(* IEC 61131-3 sources: sphere-usecases/power-hydro/implementations/openplc/st, 2 files *)

(* ---- ps_hydro_controller.st ---- *)
(*
 * SPHERE Power Systems - Generic Hydro Station Controller
 * IEC 61131-3 Structured Text for OpenPLC (matiec compatible)
 *
 * Control state machine for hydro power generation:
 *   IDLE -> STARTUP -> RUNNING -> SHUTDOWN -> IDLE
 *                  \-> TRIPPED (on any trip) -> IDLE (after reset)
 *
 * I/O Mapping (configured in OpenPLC web interface):
 *   HMI Inputs:
 *     in_Start_Cmd -> %IX0.0
 *     in_Stop_Cmd -> %IX0.1
 *     in_Reset_Cmd -> %IX0.2
 *     in_Mode_Auto -> %IX0.3
 *     in_Run_Enable -> %IX0.4
 *     in_Power_Setpoint -> %IW60
 *
 *   Process Inputs from Simulator (via bridge):
 *     in_Gate_Pos -> %IW70
 *     in_Res_Level -> %IW71
 *     in_Head -> %IW72
 *     in_Flow -> %IW73
 *     in_Pressure -> %IW74
 *     in_Speed_Pct -> %IW75
 *     in_Freq_Hz -> %IW76
 *     in_Power_MW -> %IW77
 *     in_Breaker_Sts -> %IX2.0
 *     in_Spill_Sts -> %IX2.1
 *
 *   Actuator Outputs to Simulator (via bridge):
 *     out_Gate_Cmd -> %QW100
 *     out_Power_Setpoint -> %QW101
 *     out_Breaker_Cmd -> %QX5.0
 *     out_Spill_Cmd -> %QX5.1
 *
 *   State Outputs to HMI:
 *     out_State_Idle -> %QX7.0
 *     out_State_Startup -> %QX7.1
 *     out_State_Running -> %QX7.2
 *     out_State_Shutdown -> %QX7.3
 *     out_State_Tripped -> %QX7.4
 *     out_Permissives_Ready -> %QX7.5
 *
 *   Trip Outputs:
 *     out_Trip_Overspeed -> %QX8.0
 *     out_Trip_Overpressure -> %QX8.1
 *     out_Trip_LowHead -> %QX8.2
 *     out_Trip_Manual -> %QX8.3
 *
 *   Alarm Outputs:
 *     out_Alarm_GateMismatch -> %QX9.0
 *     out_Alarm_BreakerMismatch -> %QX9.1
 *     out_Alarm_LowLevel -> %QX9.2
 *)

PROGRAM HydroController
  VAR_INPUT
    (* HMI Inputs *)
    in_Start_Cmd : BOOL;              (* Start pushbutton *)
    in_Stop_Cmd : BOOL;               (* Stop pushbutton *)
    in_Reset_Cmd : BOOL;              (* Trip reset pushbutton *)
    in_Mode_Auto : BOOL;              (* Auto mode enable *)
    in_Run_Enable : BOOL;             (* Run permissive *)
    in_Power_Setpoint : INT;          (* 0-1000 = 0-100 MW *)

    (* Process Inputs from Simulator *)
    in_Gate_Pos : INT;                (* Gate position 0-1000 = 0-100% *)
    in_Res_Level : INT;               (* Reservoir level 0-3000 = 0-30.00 m *)
    in_Head : INT;                    (* Head 0-1500 = 0-150.0 m *)
    in_Flow : INT;                    (* Flow 0-1500 = 0-150.0 m3/s *)
    in_Pressure : INT;                (* Pressure kPa *)
    in_Speed_Pct : INT;               (* Speed 0-1500 = 0-150.0% *)
    in_Freq_Hz : INT;                 (* Frequency 5500-6500 = 55-65 Hz *)
    in_Power_MW : INT;                (* Power 0-1000 = 0-100 MW *)
    in_Breaker_Sts : BOOL;            (* Breaker closed status *)
    in_Spill_Sts : BOOL;              (* Spillway open status *)
  END_VAR

  VAR_OUTPUT
    (* Actuator Outputs to Simulator *)
    out_Gate_Cmd : INT;               (* Gate command 0-1000 = 0-100% *)
    out_Power_Setpoint : INT;         (* Power setpoint passthrough *)
    out_Breaker_Cmd : BOOL;           (* Breaker close command *)
    out_Spill_Cmd : BOOL;             (* Spillway open command *)

    (* State Outputs to HMI *)
    out_State_Idle : BOOL;
    out_State_Startup : BOOL;
    out_State_Running : BOOL;
    out_State_Shutdown : BOOL;
    out_State_Tripped : BOOL;
    out_Permissives_Ready : BOOL;

    (* Trip Outputs *)
    out_Trip_Overspeed : BOOL;
    out_Trip_Overpressure : BOOL;
    out_Trip_LowHead : BOOL;
    out_Trip_Manual : BOOL;

    (* Alarm Outputs *)
    out_Alarm_GateMismatch : BOOL;
    out_Alarm_BreakerMismatch : BOOL;
    out_Alarm_LowLevel : BOOL;
  END_VAR

  VAR
    (* State Machine - 0=IDLE, 1=STARTUP, 2=RUNNING, 3=SHUTDOWN, 4=TRIPPED *)
    State : INT := 0;
    STATE_IDLE : INT := 0;
    STATE_STARTUP : INT := 1;
    STATE_RUNNING : INT := 2;
    STATE_SHUTDOWN : INT := 3;
    STATE_TRIPPED : INT := 4;

    (* Permissives *)
    Perm_Level_OK : BOOL := FALSE;
    Perm_Head_OK : BOOL := FALSE;
    Perm_No_Trips : BOOL := FALSE;
    Perm_Run_Enable : BOOL := FALSE;
    All_Permissives : BOOL := FALSE;

    (* Trip Latches *)
    Trip_Overspeed_Latch : BOOL := FALSE;
    Trip_Overpressure_Latch : BOOL := FALSE;
    Trip_LowHead_Latch : BOOL := FALSE;
    Trip_Manual_Latch : BOOL := FALSE;
    Any_Trip : BOOL := FALSE;

    (* Control Parameters *)
    No_Load_Gate_Pct : REAL := 5.0;
    Sync_Speed_Low : REAL := 99.0;
    Sync_Speed_High : REAL := 101.0;
    Min_Power_MW : REAL := 1.0;
    Kp_Gate : REAL := 2.0;
    Gate_Shutdown_Rate : REAL := 5.0;
    Gate_Emerg_Rate : REAL := 20.0;

    (* Trip Thresholds *)
    Overspeed_Trip_Pct : REAL := 110.0;
    Overpressure_Trip_kPa : REAL := 1500.0;
    Min_Head_m : REAL := 10.0;
    Low_Level_m : REAL := 8.0;

    (* Mismatch Alarm Parameters *)
    Gate_Mismatch_Pct : REAL := 5.0;
    Gate_Mismatch_Delay : INT := 50;
    Breaker_Mismatch_Delay : INT := 5;
    Gate_Mismatch_Timer : INT := 0;
    Breaker_Mismatch_Timer : INT := 0;

    (* Process Values (scaled) *)
    Gate_Pos_Pct : REAL;
    Gate_Cmd_Pct : REAL := 0.0;
    Res_Level_m : REAL;
    Head_m : REAL;
    Flow_m3s : REAL;
    Pressure_kPa : REAL;
    Speed_Pct : REAL;
    Freq_Hz : REAL;
    Power_MW : REAL;
    Power_Setpoint_MW : REAL;

    (* Control Calculations *)
    Power_Error : REAL;
    Gate_Adjustment : REAL;
    Gate_Error : REAL;

    (* Edge Detection *)
    Start_Cmd_Prev : BOOL := FALSE;
    Stop_Cmd_Prev : BOOL := FALSE;
    Reset_Cmd_Prev : BOOL := FALSE;
    Start_Rising : BOOL := FALSE;
    Stop_Rising : BOOL := FALSE;
    Reset_Rising : BOOL := FALSE;
  END_VAR

  (* 1. SCALE INPUTS *)
  Gate_Pos_Pct := INT_TO_REAL(in_Gate_Pos) / 10.0;
  Res_Level_m := INT_TO_REAL(in_Res_Level) / 100.0;
  Head_m := INT_TO_REAL(in_Head) / 10.0;
  Flow_m3s := INT_TO_REAL(in_Flow) / 10.0;
  Pressure_kPa := INT_TO_REAL(in_Pressure);
  Speed_Pct := INT_TO_REAL(in_Speed_Pct) / 10.0;
  Freq_Hz := INT_TO_REAL(in_Freq_Hz) / 100.0;
  Power_MW := INT_TO_REAL(in_Power_MW) / 10.0;
  Power_Setpoint_MW := INT_TO_REAL(in_Power_Setpoint) / 10.0;

  (* 2. EDGE DETECTION FOR COMMANDS *)
  Start_Rising := in_Start_Cmd AND NOT Start_Cmd_Prev;
  Stop_Rising := in_Stop_Cmd AND NOT Stop_Cmd_Prev;
  Reset_Rising := in_Reset_Cmd AND NOT Reset_Cmd_Prev;
  Start_Cmd_Prev := in_Start_Cmd;
  Stop_Cmd_Prev := in_Stop_Cmd;
  Reset_Cmd_Prev := in_Reset_Cmd;

  (* 3. TRIP DETECTION *)
  IF Speed_Pct > Overspeed_Trip_Pct THEN
    Trip_Overspeed_Latch := TRUE;
  END_IF;

  IF Pressure_kPa > Overpressure_Trip_kPa THEN
    Trip_Overpressure_Latch := TRUE;
  END_IF;

  IF Head_m < Min_Head_m AND State = STATE_RUNNING THEN
    Trip_LowHead_Latch := TRUE;
  END_IF;

  Any_Trip := Trip_Overspeed_Latch OR Trip_Overpressure_Latch OR
              Trip_LowHead_Latch OR Trip_Manual_Latch;

  (* 4. PERMISSIVE CHECKS *)
  Perm_Level_OK := Res_Level_m > Low_Level_m;
  Perm_Head_OK := Head_m >= Min_Head_m;
  Perm_No_Trips := NOT Any_Trip;
  Perm_Run_Enable := in_Run_Enable;

  All_Permissives := Perm_Level_OK AND Perm_Head_OK AND
                     Perm_No_Trips AND Perm_Run_Enable;

  (* 5. STATE MACHINE *)
  CASE State OF

    0: (* STATE_IDLE *)
      Gate_Cmd_Pct := 0.0;
      out_Breaker_Cmd := FALSE;
      out_Spill_Cmd := FALSE;

      IF Start_Rising AND All_Permissives THEN
        State := STATE_STARTUP;
      END_IF;

    1: (* STATE_STARTUP *)
      IF Gate_Cmd_Pct < No_Load_Gate_Pct THEN
        Gate_Cmd_Pct := Gate_Cmd_Pct + 1.0;
      ELSE
        Gate_Cmd_Pct := No_Load_Gate_Pct;
      END_IF;

      IF Speed_Pct >= Sync_Speed_Low AND Speed_Pct <= Sync_Speed_High THEN
        out_Breaker_Cmd := TRUE;
        IF in_Breaker_Sts THEN
          State := STATE_RUNNING;
        END_IF;
      END_IF;

      IF Any_Trip THEN
        State := STATE_TRIPPED;
      END_IF;

      IF Stop_Rising THEN
        State := STATE_SHUTDOWN;
      END_IF;

    2: (* STATE_RUNNING *)
      Power_Error := Power_Setpoint_MW - Power_MW;
      Gate_Adjustment := Kp_Gate * Power_Error;
      Gate_Cmd_Pct := Gate_Cmd_Pct + Gate_Adjustment;

      IF Gate_Cmd_Pct < 0.0 THEN
        Gate_Cmd_Pct := 0.0;
      END_IF;
      IF Gate_Cmd_Pct > 100.0 THEN
        Gate_Cmd_Pct := 100.0;
      END_IF;

      out_Breaker_Cmd := TRUE;

      IF Any_Trip THEN
        State := STATE_TRIPPED;
      END_IF;

      IF Stop_Rising THEN
        State := STATE_SHUTDOWN;
      END_IF;

    3: (* STATE_SHUTDOWN *)
      Gate_Cmd_Pct := Gate_Cmd_Pct - Gate_Shutdown_Rate;
      IF Gate_Cmd_Pct < 0.0 THEN
        Gate_Cmd_Pct := 0.0;
      END_IF;

      IF Power_MW < Min_Power_MW THEN
        out_Breaker_Cmd := FALSE;
      END_IF;

      IF Gate_Cmd_Pct <= 0.0 AND NOT in_Breaker_Sts THEN
        State := STATE_IDLE;
      END_IF;

      IF Any_Trip THEN
        State := STATE_TRIPPED;
      END_IF;

    4: (* STATE_TRIPPED *)
      out_Breaker_Cmd := FALSE;

      Gate_Cmd_Pct := Gate_Cmd_Pct - Gate_Emerg_Rate;
      IF Gate_Cmd_Pct < 0.0 THEN
        Gate_Cmd_Pct := 0.0;
      END_IF;

      IF Trip_Overspeed_Latch THEN
        out_Spill_Cmd := TRUE;
      END_IF;

      IF Reset_Rising AND Gate_Cmd_Pct <= 0.0 AND NOT in_Breaker_Sts THEN
        Trip_Overspeed_Latch := FALSE;
        Trip_Overpressure_Latch := FALSE;
        Trip_LowHead_Latch := FALSE;
        Trip_Manual_Latch := FALSE;
        out_Spill_Cmd := FALSE;
        State := STATE_IDLE;
      END_IF;

  END_CASE;

  (* 6. MISMATCH ALARM LOGIC *)
  Gate_Error := Gate_Cmd_Pct - Gate_Pos_Pct;
  IF Gate_Error < 0.0 THEN
    Gate_Error := -Gate_Error;
  END_IF;
  IF Gate_Error > Gate_Mismatch_Pct THEN
    Gate_Mismatch_Timer := Gate_Mismatch_Timer + 1;
    IF Gate_Mismatch_Timer >= Gate_Mismatch_Delay THEN
      out_Alarm_GateMismatch := TRUE;
    END_IF;
  ELSE
    Gate_Mismatch_Timer := 0;
    out_Alarm_GateMismatch := FALSE;
  END_IF;

  IF out_Breaker_Cmd <> in_Breaker_Sts THEN
    Breaker_Mismatch_Timer := Breaker_Mismatch_Timer + 1;
    IF Breaker_Mismatch_Timer >= Breaker_Mismatch_Delay THEN
      out_Alarm_BreakerMismatch := TRUE;
    END_IF;
  ELSE
    Breaker_Mismatch_Timer := 0;
    out_Alarm_BreakerMismatch := FALSE;
  END_IF;

  out_Alarm_LowLevel := Res_Level_m < Low_Level_m;

  (* 7. WRITE OUTPUTS *)
  out_Gate_Cmd := REAL_TO_INT(Gate_Cmd_Pct * 10.0);
  out_Power_Setpoint := in_Power_Setpoint;

  out_State_Idle := (State = STATE_IDLE);
  out_State_Startup := (State = STATE_STARTUP);
  out_State_Running := (State = STATE_RUNNING);
  out_State_Shutdown := (State = STATE_SHUTDOWN);
  out_State_Tripped := (State = STATE_TRIPPED);
  out_Permissives_Ready := All_Permissives;

  out_Trip_Overspeed := Trip_Overspeed_Latch;
  out_Trip_Overpressure := Trip_Overpressure_Latch;
  out_Trip_LowHead := Trip_LowHead_Latch;
  out_Trip_Manual := Trip_Manual_Latch;

END_PROGRAM

(* ---- ps_hydro_simulator.st ---- *)
(*
 * SPHERE Power Systems - Generic Hydro Station Simulator
 * IEC 61131-3 Structured Text for OpenPLC (matiec compatible)
 *
 * Physics model for hydro power generation:
 *   Reservoir -> Penstock -> Wicket Gate -> Turbine -> Generator -> Breaker -> Grid
 *
 * I/O Mapping (configured in OpenPLC web interface):
 *   Inputs from Controller (via bridge):
 *     in_Gate_Cmd -> %IW200
 *     in_Breaker_Cmd -> %IX3.0
 *     in_Spill_Cmd -> %IX3.1
 *
 *   Outputs to Controller (via bridge):
 *     out_Gate_Pos -> %QW300
 *     out_Res_Level -> %QW301
 *     out_Head -> %QW302
 *     out_Flow -> %QW303
 *     out_Pressure -> %QW304
 *     out_Speed_Pct -> %QW305
 *     out_Freq_Hz -> %QW306
 *     out_Power_MW -> %QW307
 *     out_Breaker_Sts -> %QX40.0
 *     out_Spill_Sts -> %QX40.1
 *)

PROGRAM HydroSimulator
  VAR_INPUT
    (* Inputs from Controller via bridge *)
    in_Gate_Cmd : INT;                (* Gate command 0-1000 = 0-100% *)
    in_Breaker_Cmd : BOOL;            (* Breaker close command *)
    in_Spill_Cmd : BOOL;              (* Spillway open command *)
  END_VAR

  VAR_OUTPUT
    (* Outputs to Controller via bridge *)
    out_Gate_Pos : INT;               (* Gate position 0-1000 = 0-100% *)
    out_Res_Level : INT;              (* Reservoir level 0-3000 = 0-30.00 m *)
    out_Head : INT;                   (* Head 0-1500 = 0-150.0 m *)
    out_Flow : INT;                   (* Flow 0-1500 = 0-150.0 m3/s *)
    out_Pressure : INT;               (* Pressure 0-2000 kPa *)
    out_Speed_Pct : INT;              (* Speed 0-1500 = 0-150.0% *)
    out_Freq_Hz : INT;                (* Frequency 5500-6500 = 55.00-65.00 Hz *)
    out_Power_MW : INT;               (* Power 0-1000 = 0-100.0 MW *)
    out_Breaker_Sts : BOOL;           (* Breaker closed status *)
    out_Spill_Sts : BOOL;             (* Spillway open status *)
  END_VAR

  VAR
    (* Physical Parameters *)
    Res_Area_m2 : REAL := 10000.0;
    Res_Level_m : REAL := 20.0;
    Res_Inflow_m3s : REAL := 50.0;
    Res_Min_m : REAL := 5.0;
    Res_Max_m : REAL := 25.0;
    Tailwater_m : REAL := 0.0;

    Penstock_Tau_sec : REAL := 5.0;
    Static_Head_m : REAL := 100.0;

    Q_Max_m3s : REAL := 100.0;
    Eta_Turbine : REAL := 0.90;
    K_Q : REAL := 10.0;

    Eta_Gen : REAL := 0.97;
    P_Rated_MW : REAL := 80.0;
    Inertia_H : REAL := 4.0;
    Sync_Speed_Pct : REAL := 100.0;

    Gate_Travel_sec : REAL := 10.0;
    Gate_Slew_Max : REAL := 10.0;
    Gate_Tau_sec : REAL := 1.0;
    Gate_Emerg_sec : REAL := 3.0;

    Breaker_Open_sec : REAL := 0.06;
    Breaker_Close_sec : REAL := 0.05;
    Spill_Open_sec : REAL := 5.0;

    RHO : REAL := 1000.0;
    G : REAL := 9.81;

    (* State Variables *)
    Gate_Pos_Pct : REAL := 0.0;
    Gate_Vel : REAL := 0.0;
    Flow_m3s : REAL := 0.0;
    Flow_Target_m3s : REAL := 0.0;
    Head_m : REAL := 100.0;
    Pressure_kPa : REAL := 981.0;
    Speed_Pct : REAL := 0.0;
    Freq_Hz : REAL := 0.0;
    P_Mech_MW : REAL := 0.0;
    P_Elec_MW : REAL := 0.0;

    Breaker_Closed : BOOL := FALSE;
    Breaker_Timer : REAL := 0.0;
    Spill_Open : BOOL := FALSE;
    Spill_Timer : REAL := 0.0;

    (* Intermediate Calculations *)
    Gate_Cmd_Pct : REAL;
    Gate_Error : REAL;
    dQ_dt : REAL;
    dLevel_dt : REAL;
    dSpeed_dt : REAL;
    P_Load_MW : REAL;
    Spill_Flow_m3s : REAL;
    abs_dQ_dt : REAL;

    Timestep : REAL := 0.1;

    Overspeed : BOOL := FALSE;
    Overpressure : BOOL := FALSE;
    LowHead : BOOL := FALSE;
    OverpresThreshold : REAL;
  END_VAR

  (* 1. PROCESS INPUTS *)
  Gate_Cmd_Pct := INT_TO_REAL(in_Gate_Cmd) / 10.0;

  IF Gate_Cmd_Pct < 0.0 THEN
    Gate_Cmd_Pct := 0.0;
  END_IF;
  IF Gate_Cmd_Pct > 100.0 THEN
    Gate_Cmd_Pct := 100.0;
  END_IF;

  (* 2. GATE ACTUATOR DYNAMICS *)
  Gate_Error := Gate_Cmd_Pct - Gate_Pos_Pct;
  Gate_Vel := Gate_Error / Gate_Tau_sec;

  IF Gate_Vel > Gate_Slew_Max THEN
    Gate_Vel := Gate_Slew_Max;
  ELSIF Gate_Vel < -Gate_Slew_Max THEN
    Gate_Vel := -Gate_Slew_Max;
  END_IF;

  Gate_Pos_Pct := Gate_Pos_Pct + Gate_Vel * Timestep;

  IF Gate_Pos_Pct < 0.0 THEN
    Gate_Pos_Pct := 0.0;
  END_IF;
  IF Gate_Pos_Pct > 100.0 THEN
    Gate_Pos_Pct := 100.0;
  END_IF;

  (* 3. RESERVOIR MASS BALANCE *)
  IF Spill_Open THEN
    IF Res_Level_m > 22.0 THEN
      Spill_Flow_m3s := 20.0 * (Res_Level_m - 22.0);
    ELSE
      Spill_Flow_m3s := 0.0;
    END_IF;
  ELSE
    Spill_Flow_m3s := 0.0;
  END_IF;

  dLevel_dt := (Res_Inflow_m3s - Flow_m3s - Spill_Flow_m3s) / Res_Area_m2;
  Res_Level_m := Res_Level_m + dLevel_dt * Timestep;

  IF Res_Level_m < 0.0 THEN
    Res_Level_m := 0.0;
  END_IF;
  IF Res_Level_m > Res_Max_m THEN
    Res_Level_m := Res_Max_m;
  END_IF;

  Head_m := Res_Level_m + Static_Head_m - Tailwater_m;
  IF Head_m < 0.0 THEN
    Head_m := 0.0;
  END_IF;

  (* 4. PENSTOCK FLOW DYNAMICS *)
  IF Head_m > 0.0 THEN
    Flow_Target_m3s := K_Q * (Gate_Pos_Pct / 100.0) * SQRT(Head_m);
  ELSE
    Flow_Target_m3s := 0.0;
  END_IF;

  IF Flow_Target_m3s > Q_Max_m3s THEN
    Flow_Target_m3s := Q_Max_m3s;
  END_IF;

  dQ_dt := (Flow_Target_m3s - Flow_m3s) / Penstock_Tau_sec;
  Flow_m3s := Flow_m3s + dQ_dt * Timestep;

  IF Flow_m3s < 0.0 THEN
    Flow_m3s := 0.0;
  END_IF;

  Pressure_kPa := RHO * G * Head_m / 1000.0;

  abs_dQ_dt := dQ_dt;
  IF abs_dQ_dt < 0.0 THEN
    abs_dQ_dt := -abs_dQ_dt;
  END_IF;
  IF abs_dQ_dt > 20.0 THEN
    Pressure_kPa := Pressure_kPa * 1.5;
  END_IF;

  (* 5. TURBINE/GENERATOR DYNAMICS *)
  P_Mech_MW := RHO * G * Flow_m3s * Head_m * Eta_Turbine / 1000000.0;

  IF Breaker_Closed THEN
    Speed_Pct := 100.0;
    Freq_Hz := 60.0;

    P_Elec_MW := P_Mech_MW * Eta_Gen;
    IF P_Elec_MW > P_Rated_MW THEN
      P_Elec_MW := P_Rated_MW;
    END_IF;
  ELSE
    IF Flow_m3s > 0.1 THEN
      dSpeed_dt := (P_Mech_MW / (P_Rated_MW * 0.1) - Speed_Pct / 50.0) / Inertia_H;
      Speed_Pct := Speed_Pct + dSpeed_dt * Timestep;
    ELSE
      dSpeed_dt := -Speed_Pct / (Inertia_H * 10.0);
      Speed_Pct := Speed_Pct + dSpeed_dt * Timestep;
    END_IF;

    IF Speed_Pct < 0.0 THEN
      Speed_Pct := 0.0;
    END_IF;
    IF Speed_Pct > 150.0 THEN
      Speed_Pct := 150.0;
    END_IF;

    Freq_Hz := 60.0 * Speed_Pct / 100.0;
    P_Elec_MW := 0.0;
  END_IF;

  (* 6. BREAKER DYNAMICS *)
  IF in_Breaker_Cmd AND NOT Breaker_Closed THEN
    Breaker_Timer := Breaker_Timer + Timestep;
    IF Breaker_Timer >= Breaker_Close_sec THEN
      IF Speed_Pct >= 99.0 AND Speed_Pct <= 101.0 THEN
        Breaker_Closed := TRUE;
      END_IF;
      Breaker_Timer := 0.0;
    END_IF;
  ELSIF NOT in_Breaker_Cmd AND Breaker_Closed THEN
    Breaker_Timer := Breaker_Timer + Timestep;
    IF Breaker_Timer >= Breaker_Open_sec THEN
      Breaker_Closed := FALSE;
      Breaker_Timer := 0.0;
    END_IF;
  ELSE
    Breaker_Timer := 0.0;
  END_IF;

  (* 7. SPILLWAY DYNAMICS *)
  IF in_Spill_Cmd AND NOT Spill_Open THEN
    Spill_Timer := Spill_Timer + Timestep;
    IF Spill_Timer >= Spill_Open_sec THEN
      Spill_Open := TRUE;
      Spill_Timer := 0.0;
    END_IF;
  ELSIF NOT in_Spill_Cmd AND Spill_Open THEN
    Spill_Timer := Spill_Timer + Timestep;
    IF Spill_Timer >= Spill_Open_sec THEN
      Spill_Open := FALSE;
      Spill_Timer := 0.0;
    END_IF;
  ELSE
    Spill_Timer := 0.0;
  END_IF;

  (* 8. TRIP CONDITION DETECTION *)
  Overspeed := Speed_Pct > 110.0;
  OverpresThreshold := (RHO * G * Static_Head_m / 1000.0) * 1.5;
  Overpressure := Pressure_kPa > OverpresThreshold;
  LowHead := Head_m < 10.0;

  (* 9. WRITE OUTPUTS *)
  out_Gate_Pos := REAL_TO_INT(Gate_Pos_Pct * 10.0);
  out_Res_Level := REAL_TO_INT(Res_Level_m * 100.0);
  out_Head := REAL_TO_INT(Head_m * 10.0);
  out_Flow := REAL_TO_INT(Flow_m3s * 10.0);
  out_Pressure := REAL_TO_INT(Pressure_kPa);
  out_Speed_Pct := REAL_TO_INT(Speed_Pct * 10.0);
  out_Freq_Hz := REAL_TO_INT(Freq_Hz * 100.0);
  out_Power_MW := REAL_TO_INT(P_Elec_MW * 10.0);

  out_Breaker_Sts := Breaker_Closed;
  out_Spill_Sts := Spill_Open;

END_PROGRAM
